Staubli VAL3: setTrajItem.pgx

public program setTrajItem(TrajectoryItem& x_tTraj[] (dimensions=1), num x_nIndex (dimensions=1))
begin
  //
  // set all the field
  //
  pEditPoint.tData[x_nIndex].tSuper=x_tTraj
  // active the save data
  bToSave=true
end
